// TIA Portal V21 program export: 1 tag tables, 0 data types, 0 data blocks, 2 code blocks (in call order from the OBs), 0 instance data blocks

VAR_GLOBAL   // PLC tag table "Default tag table"
   Start AT %I0.0 : Bool;
   Stop AT %I0.1 : Bool;
   Run AT %M0.0 : Bool;
END_VAR

ORGANIZATION_BLOCK "Main"   // OB1, LAD, ProgramCycle
TITLE = "Main Program Sweep (Cycle)"
{ S7_Optimized_Access := 'TRUE' }
// stored: SetENOAutomatically false
   VAR_INPUT
      Initial_Call : Bool;   // Initial call of this OB
      Remanence : Bool;   // =True, if remanent data are available
   END_VAR
BEGIN

REGION Network 1
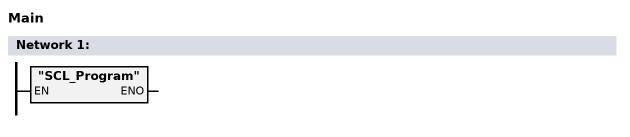
   RUNG wire#powerrail
      "SCL_Program"()
   END_RUNG
   // the same network as SCL:
   "SCL_Program"();
END_REGION
END_ORGANIZATION_BLOCK

FUNCTION "SCL_Program" : Void
{ S7_Optimized_Access := 'TRUE' }
VERSION : 0.1

BEGIN
	
	IF "Stop" THEN
	    "Run" := FALSE;   // Stop
	ELSIF "Start" THEN
	    "Run" := TRUE;    // Start
	END_IF;
	
END_FUNCTION
